INTERFACE IPistonVertical

METHOD MoveDown : TcoCore.ITcoTaskStatus
END_METHOD

METHOD MoveUp : TcoCore.ITcoTaskStatus
END_METHOD

END_INTERFACE

(* stored: Version 1.1.0.1, ProductVersion 3.1.4024.6
   Itf IPistonVertical: Id {003657db-44c8-4937-9725-21539bc48697}
   Folder Vertical: Id {4facddc6-6e42-4882-8021-7f7b480dc0ca}
   Method MoveDown: Id {abaea21b-f9f5-4a18-962b-d90095d4494e}
   Method MoveUp: Id {f45520a0-c451-49de-a144-c9529b544a47} *)
